{attribute 'qualified_only'}
VAR_GLOBAL
    fbArbiter: FB_Arbiter(1);
    fbFastFaultOutput1: FB_HardwareFFOutput := (bAutoReset := TRUE, i_sNetID := '172.21.148.148.1.1');
END_VAR

(* stored: Version 1.1.0.1
   GVL GVL: Id {9b9d6ea6-28e0-43fe-bc83-62be23c2a739} *)
